// TwinCAT 3 PLC project Coneying
// ProgramVersion: 3.1.4024.0
// libraries:
//   Tc2_Math, * (Beckhoff Automation GmbH)
//   Tc2_SPA, * (Beckhoff Automation GmbH)
//   Tc2_Standard, * (Beckhoff Automation GmbH)
//   Tc2_System, * (Beckhoff Automation GmbH)
//   Tc2_Utilities, * (Beckhoff Automation GmbH)
//   Tc3_Module, * (Beckhoff Automation GmbH)
// project tree:
//   GVLs/ Random.TcGVL
//   / PlcTask.TcTTO
//   POUs/ FB_OrangeConveyor.TcPOU, FB_LTU_Cylinder.TcPOU, FB_Reader.TcPOU, FB_Route12to6.TcPOU, FB_Route12to9.TcPOU, FB_Route3to12.TcPOU, FB_Route3to6.TcPOU, FB_Route3to9.TcPOU, FB_Route9to12.TcPOU, FB_Route6to3.TcPOU, FB_Route6to9.TcPOU, FB_Route6to12.TcPOU, FB_Route9to6.TcPOU, FB_Route9to3.TcPOU, MAIN.TcPOU, FB_ConveyorMotor.TcPOU, FB_GreenConveyor.TcPOU, Reader.TcPOU, FB_Stopper.TcPOU, FB_Route12to3.TcPOU
// real-time tasks:
//   TASK PlcTask: cycle T#30ms, priority 20, ADS port 350

CONFIGURATION Coneying
    RESOURCE PLC ON TwinCAT3
        TASK PlcTask(INTERVAL := T#30ms, PRIORITY := 20);
        PROGRAM MAIN WITH PlcTask : MAIN;
    END_RESOURCE
END_CONFIGURATION

// ---- GVLs/Random.TcGVL
{attribute 'qualified_only'}
VAR_GLOBAL
	number:int:=0;
	i: INT:=0;
END_VAR

// ---- POUs/MAIN.TcPOU
PROGRAM MAIN
VAR
	fbReader			:FB_Reader;
	fbRoute3to6			:FB_Route3to6;
	fbRoute3to9			:FB_Route3to9;
	fbRoute3to12		:FB_Route3to12;
	fbRoute6to3			:FB_Route6to3;
	fbRoute6to9			:FB_Route6to9;
	fbRoute6to12		:FB_Route6to12;
	fbRoute9to3			:FB_Route9to3;
	fbRoute9to6			:FB_Route9to6;
	fbRoute9to12		:FB_Route9to12;
	fbRoute12to3		:FB_Route12to3;
	fbRoute12to6		:FB_Route12to6;
	fbRoute12to9		:FB_Route12to9;
END_VAR

Reader();	
fbRoute3to6();		
fbRoute3to9();			
fbRoute3to12();		
fbRoute6to3();		
fbRoute6to9();		
fbRoute6to12();	
fbRoute9to3	();
fbRoute9to6();
fbRoute9to12();	
fbRoute12to3();		
fbRoute12to6();		
fbRoute12to9();

END_PROGRAM

// ---- POUs/FB_Reader.TcPOU
FUNCTION_BLOCK FB_Reader
VAR
	numbers : ARRAY[1..5] OF INT := [12, 3, 6, 9,0];  // Your set of numbers
    randomIndex 	: LREAL;
	correctIndex	: INT;
    // 	: INT;
	DRAND			: DRAND;
	
END_VAR
VAR_OUTPUT
	randomNumber: INT;
END_VAR

DRAND(SEED:=0,Num=>randomIndex);
correctIndex:= LREAL_TO_INT(randomIndex*5);
randomNumber := numbers[correctIndex];

END_FUNCTION_BLOCK

// ---- POUs/FB_Route3to6.TcPOU
FUNCTION_BLOCK FB_Route3to6
VAR
	GreenRight	:FB_GreenConveyor;				//Right Green Conveyor
	GreenLeft	:FB_GreenConveyor;				//Left Green Conveyor
	OrangeUpper	:FB_OrangeConveyor;				//Upper Orange Conveyor
	OrangeLower	:FB_OrangeConveyor;				//Lower Orange Conveyor
	nStatus: INT;
END_VAR

CASE nStatus OF
0:	OrangeLower.Motor.RunMotor();
	//Reader();
	IF Random.number=6 THEN
		nStatus:=10;
	END_IF
	10:	IF  OrangeLower.LTU.Occupied THEN					//chConveyot_GL.upied
			OrangeLower.BlueStopper.MoveStopper();			//If occupied move stopper
			nStatus:=20;
			ELSE
			OrangeLower.LTU.MoveBottom();					//LTU Move bottom to move on green
			nStatus:=20;									//jmp to state 10
		END_IF	
	20:	nStatus:=0;
END_CASE

END_FUNCTION_BLOCK

// ---- POUs/FB_GreenConveyor.TcPOU
FUNCTION_BLOCK FB_GreenConveyor
VAR
	Motor					:FB_ConveyorMotor;
	LTU						:FB_LTU_Cylinder;	
    BlueStopper				:FB_Stopper;
    nStatus					:INT:=0;	
				
END_VAR

END_FUNCTION_BLOCK

// ---- POUs/FB_ConveyorMotor.TcPOU
FUNCTION_BLOCK FB_ConveyorMotor
VAR
	bStart			AT%Q*		:BOOL;	//Output to turn motor on
	bFuse			AT%I*		:BOOL;	//Motor is Running
	bThermistor		AT%I*		:BOOL;	//Motor is Ok
END_VAR

PROPERTY Fuse : BOOL
GET
Fuse:=bFuse;
END_GET
END_PROPERTY

METHOD RunMotor : BOOL
VAR
	Motor	:FB_ConveyorMotor;
END_VAR
IF Motor.bStart AND NOT FUSE AND NOT Thermistor THEN
	RunMotor:=TRUE;
	ELSE
	RunMotor:=FALSE;
END_IF
END_METHOD

PROPERTY Start : BOOL
SET
bStart:=Start;
END_SET
END_PROPERTY

PROPERTY Thermistor : BOOL
GET
Thermistor:=bThermistor;
END_GET
END_PROPERTY

END_FUNCTION_BLOCK

// ---- POUs/FB_LTU_Cylinder.TcPOU
FUNCTION_BLOCK FB_LTU_Cylinder
VAR
		bLightBarrier	AT %I*			: BOOL;				// LTU light sensor 
		bToBottom		AT %Q* 			: BOOL; 			// Output TO Bottom	
		bToTop			AT %Q* 			: BOOL; 			// Output To Top
		bAtBottom		AT %I*			: BOOL; 			//Input At Bottom 
		bAtMiddle 		AT %I* 			: BOOL; 			//Input At Middle	 
		bAtTop			AT %I* 			: BOOL; 			//Input At Top 
		LTU_Motor						: FB_ConveyorMotor;	//LTU Motor
END_VAR

PROPERTY AtBottom : BOOL
GET
AtBottom:= bAtBottom;
END_GET
END_PROPERTY

PROPERTY AtMiddle : BOOL
GET
AtMiddle:= bAtMiddle;
END_GET
END_PROPERTY

PROPERTY AtTop : BOOL
GET
AtTop:= bAtTop;
END_GET
END_PROPERTY

METHOD MoveBottom : BOOL
VAR
	Cylinder	:FB_LTU_Cylinder;
END_VAR
IF NOT Cylinder.Occupied THEN
Cylinder.ToBottom	:=TRUE; 	// Set Output To bottom to True 
Cylinder.ToTop	:=FALSE;		// Set Output To Top to FALSE
END_IF
IF NOT Cylinder.AtTop AND Cylinder.AtBottom AND NOT Cylinder.AtMiddle THEN //Check the feedback inputs
	MoveBottom:=TRUE;			//return true
	ELSE
		MoveBottom:=FALSE;		//return false
END_IF
END_METHOD

METHOD MoveMiddle : BOOL
VAR
	Cylinder	:FB_LTU_Cylinder;
END_VAR
IF NOT Cylinder.Occupied THEN
Cylinder.ToBottom	:=FALSE; 	// Set Output To bottom to false 
Cylinder.ToTop	:=FALSE;		// Set Output To Top to false
END_IF
IF NOT Cylinder.AtTop AND NOT Cylinder.AtBottom AND Cylinder.AtMiddle THEN //Check the feedback inputs
	MoveMiddle:=TRUE;			//return true
	ELSE
		MoveMiddle:=FALSE;		//return false
END_IF
END_METHOD

METHOD MoveTop : BOOL
VAR
	Cylinder	:FB_LTU_Cylinder;
END_VAR
IF NOT Cylinder.Occupied THEN
Cylinder.ToBottom	:=FALSE; 	// Set Output To bottom to false 
Cylinder.ToTop	:=TRUE;		// Set Output To Top to True
END_IF
IF Cylinder.AtTop AND NOT Cylinder.AtBottom AND NOT Cylinder.AtMiddle THEN
	MoveTop:=TRUE;
	ELSE
		MoveTop:=FALSE;
END_IF
END_METHOD

PROPERTY Occupied : BOOL
GET
Occupied:= bLightBarrier;
END_GET
END_PROPERTY

PROPERTY ToBottom : BOOL
SET
bToBottom:=ToBottom ;
END_SET
END_PROPERTY

PROPERTY ToTop : BOOL
SET
bToTop:=ToTop;
END_SET
END_PROPERTY

END_FUNCTION_BLOCK

// ---- POUs/FB_Stopper.TcPOU
FUNCTION_BLOCK FB_Stopper
VAR
	bStopperCylinder		AT%Q*		: BOOL; //Cylinder moves stopper down
	bStopperSensor			AT%I*		: BOOL; //Sensor checks if stopper is occupied
END_VAR

METHOD MoveStopper : BOOL
VAR
	Stopper:FB_Stopper;
END_VAR
IF NOT Stopper.Occupied THEN			//If stopper is nor occupied
	Stopper.StopperCylinder:=TRUE;		//Move stopper up
END_IF
END_METHOD

PROPERTY Occupied : BOOL
GET
Occupied:=bStopperSensor;
END_GET
END_PROPERTY

PROPERTY StopperCylinder : BOOL
SET
bStopperCylinder:=StopperCylinder;
END_SET
END_PROPERTY

METHOD StopperDown : BOOL
VAR
	Stopper:FB_Stopper;
END_VAR
IF NOT Stopper.Occupied THEN			//If stopper is nor occupied
	Stopper.StopperCylinder:=FALSE;		//Move stopper up
END_IF
END_METHOD

END_FUNCTION_BLOCK

// ---- POUs/FB_OrangeConveyor.TcPOU
FUNCTION_BLOCK FB_OrangeConveyor
VAR
	Motor					:FB_ConveyorMotor;
	LTU						:FB_LTU_Cylinder;	
    BlueStopper				:FB_Stopper;
	PurpleStopper_1			:FB_Stopper;
	PurpleStopper_2			:FB_Stopper;
    nStatus					:INT:=0;					
END_VAR

END_FUNCTION_BLOCK

// ---- POUs/FB_Route3to9.TcPOU
FUNCTION_BLOCK FB_Route3to9
VAR
	GreenRight	:FB_GreenConveyor;				//Right Green Conveyor
	GreenLeft	:FB_GreenConveyor;				//Left Green Conveyor
	OrangeUpper	:FB_OrangeConveyor;				//Upper Orange Conveyor
	OrangeLower	:FB_OrangeConveyor;				//Lower Orange Conveyor
	nStatus: INT;
END_VAR

CASE nStatus OF
0:	OrangeLower.Motor.RunMotor();
	//Reader();
	IF Random.number=9 THEN
	nStatus:=10;
END_IF
10:	IF  OrangeLower.LTU.Occupied THEN					//chConveyot_GL.upied
		OrangeLower.BlueStopper.MoveStopper();			//If occupied move stopper
		nStatus:=20;
		ELSE
		OrangeLower.LTU.MoveTop();					//LTU Move Top to saty on Orange
		nStatus:=20;									//jmp to state 10
	END_IF										
20:	IF GreenLeft.LTU.Occupied THEN							//check LTU occupied
				OrangeLower.PurpleStopper_1.MoveStopper();		
				ELSE
				OrangeLower.PurpleStopper_2.StopperDown();	
				GreenLeft.LTU.MoveTop();			//LTU Move Top to move on orange
				nStatus:=30;
			END_IF
30:	nStatus:=0;
END_CASE

END_FUNCTION_BLOCK

// ---- POUs/FB_Route3to12.TcPOU
FUNCTION_BLOCK FB_Route3to12
VAR
	GreenRight	:FB_GreenConveyor;				//Right Green Conveyor
	GreenLeft	:FB_GreenConveyor;				//Left Green Conveyor
	OrangeUpper	:FB_OrangeConveyor;				//Upper Orange Conveyor
	OrangeLower	:FB_OrangeConveyor;				//Lower Orange Conveyor
	nStatus: INT;
END_VAR

CASE nStatus OF
0:	OrangeLower.Motor.RunMotor();
	//Reader();
	IF Random.number=12 THEN
	nStatus:=10;
END_IF
10:	IF  OrangeLower.LTU.Occupied THEN					//chConveyot_GL.upied
		OrangeLower.BlueStopper.MoveStopper();			//If occupied move stopper
		nStatus:=20;
		ELSE
		OrangeLower.LTU.MoveTop();					//LTU Move Top to saty on Orange
		nStatus:=20;									//jmp to state 10
	END_IF										
20:	IF GreenLeft.LTU.Occupied THEN							//check LTU occupied
				OrangeLower.PurpleStopper_1.MoveStopper();			//LTU Move bottom to saty on green
				ELSE
				OrangeLower.PurpleStopper_2.MoveStopper();
				GreenLeft.LTU.MoveTop();			//LTU Move Top to move on orange
				nStatus:=30;
			END_IF
30:	IF NOT  OrangeUpper.LTU.Occupied THEN
			GreenLeft.LTU.MoveBottom();			//LTU Move Bottom to move on green
			nStatus:=40;
	END_IF
40:	nStatus:=0;
END_CASE

END_FUNCTION_BLOCK

// ---- POUs/FB_Route6to3.TcPOU
FUNCTION_BLOCK FB_Route6to3
VAR
	GreenRight	:FB_GreenConveyor;				//Right Green Conveyor
	GreenLeft	:FB_GreenConveyor;				//Left Green Conveyor
	OrangeUpper	:FB_OrangeConveyor;				//Upper Orange Conveyor
	OrangeLower	:FB_OrangeConveyor;				//Lower Orange Conveyor
	nStatus: INT;
END_VAR

CASE nStatus OF
	0:	GreenLeft.Motor.RunMotor();
		//Reader();
	IF Random.number=3 THEN
		nStatus:=10;
	END_IF
	
	10:	IF  GreenLeft.LTU.Occupied THEN								//check LTU occupied
			 GreenLeft.BlueStopper.MoveStopper();						//If occupied move stopper
			ELSE
			GreenLeft.LTU.MoveTop();
			nStatus:=20;
		END_IF										
	20:		IF  GreenRight.LTU.Occupied THEN								//check LTU occupied
			 OrangeUpper.PurpleStopper_1.MoveStopper();						//If occupied move stopper
			ELSE
			OrangeUpper.PurpleStopper_2.StopperDown();			
			GreenRight.LTU.MoveTop();
			nStatus:=30;
		END_IF
	30:	nStatus:=0;		
END_CASE

END_FUNCTION_BLOCK

// ---- POUs/FB_Route6to9.TcPOU
FUNCTION_BLOCK FB_Route6to9
VAR
	GreenRight	:FB_GreenConveyor;				//Right Green Conveyor
	GreenLeft	:FB_GreenConveyor;				//Left Green Conveyor
	OrangeUpper	:FB_OrangeConveyor;				//Upper Orange Conveyor
	OrangeLower	:FB_OrangeConveyor;				//Lower Orange Conveyor
	nStatus: INT;
END_VAR

CASE nStatus OF
	0:	GreenLeft.Motor.RunMotor();
		//Reader();
	IF Random.number=9 THEN
		nStatus:=10;
	END_IF
	10:	IF  GreenLeft.LTU.Occupied THEN								//check LTU occupied
			 GreenLeft.BlueStopper.MoveStopper();						//If occupied move stopper
			ELSE
			GreenLeft.LTU.MoveTop();
			nStatus:=20;
		END_IF				
	20:	nStatus:=0;
END_CASE

END_FUNCTION_BLOCK

// ---- POUs/FB_Route6to12.TcPOU
FUNCTION_BLOCK FB_Route6to12
VAR
	GreenRight	:FB_GreenConveyor;				//Right Green Conveyor
	GreenLeft	:FB_GreenConveyor;				//Left Green Conveyor
	OrangeUpper	:FB_OrangeConveyor;				//Upper Orange Conveyor
	OrangeLower	:FB_OrangeConveyor;				//Lower Orange Conveyor
	nStatus: INT;
END_VAR

CASE nStatus OF
	0:	GreenLeft.Motor.RunMotor();
		//Reader();
		IF Random.number=12 THEN
		nStatus:=10;
	END_IF
	
	10:	IF  GreenLeft.LTU.Occupied THEN					//chConveyot_GL.upied
			GreenLeft.BlueStopper.MoveStopper();			//If occupied move stopper
			nStatus:=20;
			ELSE
			GreenLeft.LTU.MoveBottom();					//LTU Move bottom to saty on green
			nStatus:=20;									//jmp to state 10
		END_IF										
	20:	IF NOT OrangeUpper.LTU.Occupied THEN				//check LTU occupied
					OrangeUpper.LTU.MoveBottom();			//LTU Move bottom to saty on green
					ELSE
					GreenLeft.LTU.MoveMiddle();			//LTU Move middle to stop on green
					nStatus:=30;	
				END_IF
	30:	nStatus:=0;
END_CASE

END_FUNCTION_BLOCK

// ---- POUs/FB_Route9to3.TcPOU
FUNCTION_BLOCK FB_Route9to3
VAR
	GreenRight	:FB_GreenConveyor;				//Right Green Conveyor
	GreenLeft	:FB_GreenConveyor;				//Left Green Conveyor
	OrangeUpper	:FB_OrangeConveyor;				//Upper Orange Conveyor
	OrangeLower	:FB_OrangeConveyor;				//Lower Orange Conveyor
	nStatus: INT;
END_VAR

CASE nStatus OF
	0:	OrangeUpper.Motor.RunMotor();
		//Reader();
	IF Random.number=3 THEN
		nStatus:=10;
	END_IF
	10:	IF  OrangeUpper.LTU.Occupied THEN					//check LTU occupied
			OrangeUpper.BlueStopper.MoveStopper();			//If occupied move stopper
			nStatus:=20;
			ELSE
			OrangeLower.LTU.MoveTop();					//LTU Move Top to saty on Orange
			nStatus:=20;									//jmp to state 10
		END_IF										
	20:	IF  GreenRight.LTU.Occupied THEN							//check LTU occupied
					OrangeLower.PurpleStopper_1.MoveStopper();			//LTU Move bottom to saty on green
					ELSE
					OrangeLower.PurpleStopper_1.StopperDown();	
					GreenLeft.LTU.MoveTop();			//LTU Move Top to move on orange
					nStatus:=30;
				END_IF
	30: nStatus:=0;
END_CASE

END_FUNCTION_BLOCK

// ---- POUs/FB_Route9to6.TcPOU
FUNCTION_BLOCK FB_Route9to6
VAR
	GreenRight	:FB_GreenConveyor;				//Right Green Conveyor
	GreenLeft	:FB_GreenConveyor;				//Left Green Conveyor
	OrangeUpper	:FB_OrangeConveyor;				//Upper Orange Conveyor
	OrangeLower	:FB_OrangeConveyor;				//Lower Orange Conveyor
	nStatus: INT;
END_VAR

CASE nStatus OF
	0:	OrangeUpper.Motor.RunMotor();
		//Reader();
	IF Random.number=6 THEN
		nStatus:=10;
	END_IF
	10:	IF  OrangeUpper.LTU.Occupied THEN					//check LTU occupied
			OrangeUpper.BlueStopper.MoveStopper();			//If occupied move stopper
			nStatus:=20;
			ELSE
			OrangeUpper.LTU.MoveTop();					//LTU Move Top to saty on Orange
			nStatus:=20;									//jmp to state 10
		END_IF										
	20:	IF  GreenRight.LTU.Occupied THEN							//check LTU occupied
					OrangeUpper.PurpleStopper_1.MoveStopper();			//LTU Move bottom to saty on green
					ELSE
					OrangeUpper.PurpleStopper_1.StopperDown();	
					nStatus:=30;
				END_IF
	30: IF  OrangeLower.LTU.Occupied THEN							//check LTU occupied
					GreenRight.LTU.MoveMiddle();			//LTU Move middle to stop on green
					ELSE
					GreenRight.LTU.MoveBottom();			//LTU Move bottom to move on green
					nStatus:=40;
				END_IF
	40:	nStatus:=0;
END_CASE

END_FUNCTION_BLOCK

// ---- POUs/FB_Route9to12.TcPOU
FUNCTION_BLOCK FB_Route9to12
VAR
	GreenRight	:FB_GreenConveyor;				//Right Green Conveyor
	GreenLeft	:FB_GreenConveyor;				//Left Green Conveyor
	OrangeUpper	:FB_OrangeConveyor;				//Upper Orange Conveyor
	OrangeLower	:FB_OrangeConveyor;				//Lower Orange Conveyor
	nStatus: INT;
END_VAR

CASE nStatus OF
	0:	OrangeUpper.Motor.RunMotor();
		//Reader();
	IF Random.number=3 THEN
		nStatus:=10;
	END_IF
	10:	IF  OrangeUpper.LTU.Occupied THEN					//check LTU occupied
			OrangeUpper.BlueStopper.MoveStopper();			//If occupied move stopper
			nStatus:=20;
			ELSE
			OrangeUpper.LTU.MoveBottom();					//LTU Move Top to move on Green
			nStatus:=20;									//jmp to state 10
		END_IF										
	20: nStatus:=0;
END_CASE

END_FUNCTION_BLOCK

// ---- POUs/FB_Route12to3.TcPOU
FUNCTION_BLOCK FB_Route12to3
VAR
	nStatus		:INT	:=0;
	GreenRight	:FB_GreenConveyor;				//Right Green Conveyor
	GreenLeft	:FB_GreenConveyor;				//Left Green Conveyor
	OrangeUpper	:FB_OrangeConveyor;				//Upper Orange Conveyor
	OrangeLower	:FB_OrangeConveyor;				//Lower Orange Conveyor
END_VAR

CASE nStatus OF
0:	GreenRight.Motor.RunMotor();								//Run motor
	//Reader();
	IF Random.number=3 THEN		//check destination
	nStatus:=10;
END_IF
10:	IF GreenRight.LTU.Occupied THEN					//check LTU occupied
		GreenRight.BlueStopper.MoveStopper();			//If occupied move stopper
		ELSE
		GreenRight.LTU.MoveTop();					//LTU Move bottom to saty on green
		nStatus:=20;									
	END_IF										
20:	nStatus:=0;
END_CASE

END_FUNCTION_BLOCK

// ---- POUs/FB_Route12to6.TcPOU
FUNCTION_BLOCK FB_Route12to6
VAR
	nStatus		:INT	:=0;
	GreenRight	:FB_GreenConveyor;				//Right Green Conveyor
	GreenLeft	:FB_GreenConveyor;				//Left Green Conveyor
	OrangeUpper	:FB_OrangeConveyor;				//Upper Orange Conveyor
	OrangeLower	:FB_OrangeConveyor;				//Lower Orange Conveyor
END_VAR

CASE nStatus OF
0:	GreenRight.Motor.RunMotor();
	//Reader();
	IF Random.number=6 THEN
	nStatus:=10;
END_IF
10:	IF  GreenRight.LTU.Occupied THEN					//check LTU occupied
		GreenRight.BlueStopper.MoveStopper();			//If occupied move stopper
		ELSE
		GreenRight.LTU.MoveBottom();					//LTU Move bottom to saty on green
		nStatus:=20;									
	END_IF										
20:	IF NOT OrangeLower.LTU.Occupied THEN				//check LTU occupied
				OrangeLower.LTU.MoveBottom();			//LTU Move bottom to saty on green
				nStatus:=30;
				ELSE
				GreenRight.LTU.MoveMiddle();			//LTU Move middle to stop on green
			END_IF
30:	nStatus:=0;
END_CASE

END_FUNCTION_BLOCK

// ---- POUs/FB_Route12to9.TcPOU
FUNCTION_BLOCK FB_Route12to9
VAR
	nStatus		:INT	:=0;
	MoveBottom: INT;
	GreenRight	:FB_GreenConveyor;				//Right Green Conveyor
	GreenLeft	:FB_GreenConveyor;				//Left Green Conveyor
	OrangeUpper	:FB_OrangeConveyor;				//Upper Orange Conveyor
	OrangeLower	:FB_OrangeConveyor;				//Lower Orange Conveyor
END_VAR

CASE nStatus OF
0:	GreenRight.Motor.RunMotor();
	//Reader();
	IF Random.number=9 THEN
	nStatus:=10;
END_IF
10:	IF  GreenRight.LTU.Occupied THEN					//check LTU occupied
		GreenRight.BlueStopper.MoveStopper();			//If occupied move stopper
		ELSE
		GreenRight.LTU.MoveBottom();					//LTU Move bottom to saty on green
		nStatus:=20;									
	END_IF										
20:	IF NOT OrangeLower.LTU.Occupied THEN				//check LTU occupied
				OrangeLower.LTU.MoveTop();			//LTU Move bottom to saty on green
				nStatus:=30;
				ELSE
				GreenRight.LTU.MoveMiddle();			//LTU Move middle to stop on green
			END_IF
30:	IF NOT GreenLeft.LTU.Occupied THEN				//check LTU occupied
				OrangeLower.LTU.MoveTop();			//LTU Move bottom to saty on green
				GreenLeft.LTU.MoveTop();
				nStatus:=40;
				ELSE
				OrangeLower.PurpleStopper_1.MoveStopper();			//LTU Move middle to stop on green
			END_IF;
40:	nStatus:=0;
END_CASE

END_FUNCTION_BLOCK

// ---- POUs/Reader.TcPOU
FUNCTION Reader : INT
VAR
	numbers : ARRAY[1..5] OF INT := [12, 3, 6, 9];  // Your set of numbers
	
END_VAR

Random.number:=Random.number+3;
IF Random.number>12 THEN
	Random.number:=0;
END_IF

END_FUNCTION
